Fanuc KAREL source: NC0073.KL

-- PROVISIONAL review KL for V940-1; original PC SHA256 abf77574df8fa1881136dfb8bb280939d129e778fcf6bf5c7cdd251641489a95
-- Incomplete behavior may be omitted. Consult companion uncertainty JSON. Do not deploy.
PROGRAM NC0073
%NOLOCKGROUP
-- UNRESOLVED_LOCAL_POOL 1 cells at code offset 3; source declarations unknown
-- DIRECT_LOCAL_WORD_ACCESS alone does not prove INTEGER, REAL, or BOOLEAN
BEGIN
  -- V9_OWNER_INTERVAL_HINT [6,25),[11,23); structural only; source/VM held
  -- V9_EXPOSED_INDEXED_TABLE_HINT layout=0001; 4 counted words exposed once; source arms/runtime held
  -- UNRESOLVED_PC offsets 0-8; opcodes 2B,2C,7B
  -- UNRESOLVED_PC offsets 13-20; opcodes 9D,23
  -- UNRESOLVED_PC offsets 25-42; opcodes 21,2E,59,79
  -- UNRESOLVED_PC offsets 47-64; opcodes 21,2E,59,79
  -- UNRESOLVED_PC offsets 69-83; opcodes 21,9D,52,23
  -- UNRESOLVED_PC offsets 88-93; opcodes 7A
  -- UNRESOLVED_PC offsets 98-103; opcodes 7A
  -- UNRESOLVED_PC offsets 108-112; opcodes 7F
  -- UNRESOLVED_PC offsets 117-121; opcodes 27,AA
  -- UNRESOLVED_PC offsets 126-130; opcodes 7F
END NC0073
